// TIA Portal V20 export
TYPE "typeCmControlNodeBrakeTest"
// stored: Namespace Unit1.Em5
   STRUCT
      magazine { ExternalWritable := 'False'} : "LER_typeBrakeTestEmControlNodes";
   END_STRUCT;
END_TYPE
